FUNCTION_BLOCK FB_LimSwStatusMCS2 IMPLEMENTS I_LimSwStatusMCS2
VAR_INPUT
END_VAR
VAR_OUTPUT
END_VAR
VAR
    bPositiveDirection : BOOL;
    bNegativeDirection : BOOL;
    bMoveBackwardEnabled : BOOL;
    bMoveForwardEnabled : BOOL;
    bInternalLimitActive : BOOL;
    bWarningCondition : BOOL;
    bLimOverride : BOOL;
END_VAR

// Read Limits status and update shared space
bMoveBackwardEnabled := bLimOverride OR NOT(THIS^.bNegativeDirection AND ( THIS^.bInternalLimitActive OR THIS^.bWarningCondition ));
bMoveForwardEnabled := bLimOverride OR NOT(THIS^.bPositiveDirection AND ( THIS^.bInternalLimitActive OR THIS^.bWarningCondition ));

METHOD AxisStatus
VAR_INPUT
    PositiveDirection	: BOOL;
    NegativeDirection	: BOOL;
END_VAR
bPositiveDirection:=PositiveDirection;
bNegativeDirection:=NegativeDirection;
END_METHOD

{warning 'Add property implementation'}
PROPERTY InternalLimitActive : BOOL
GET
END_GET
SET
END_SET
END_PROPERTY

METHOD InternalLimits
VAR_INPUT
    InternalLimitActive	: BOOL;
    WarningCondition	: BOOL;
END_VAR
bInternalLimitActive := InternalLimitActive;
bWarningCondition := WarningCondition;
END_METHOD

{warning 'Add property implementation'}
PROPERTY LimBackward : BOOL
GET
END_GET
END_PROPERTY

{warning 'Add property implementation'}
PROPERTY LimForward : BOOL
GET
END_GET
END_PROPERTY

{warning 'Add property implementation'}
PROPERTY LimHome : BOOL
GET
END_GET
END_PROPERTY

{warning 'Add property implementation'}
PROPERTY LimOverride : BOOL
GET
END_GET
SET
END_SET
END_PROPERTY

{warning 'Add property implementation'}
PROPERTY MoveBackwardEnabled : BOOL
GET
END_GET
END_PROPERTY

{warning 'Add property implementation'}
PROPERTY MoveForwardEnabled : BOOL
GET
END_GET
END_PROPERTY

{warning 'Add property implementation'}
PROPERTY WarningCondition : BOOL
GET
END_GET
SET
END_SET
END_PROPERTY

END_FUNCTION_BLOCK

(* stored: Version 1.1.0.1
   POU FB_LimSwStatusMCS2: Id {e82c472b-4e09-459d-83c5-e6524de07cc9}, SpecialFunc None
   Method AxisStatus: Id {b6a43cf8-24d6-42e3-9ffa-0a6a1fcfe0c2}
   Property InternalLimitActive: Id {9785faa9-6e22-4b72-879f-74f38349c993}
   Get Get: Id {d5fc83b0-3602-4b79-b305-31cda962b007}
   Set Set: Id {3ae2133f-fa8c-4126-95ec-f568abc28cb6}
   Method InternalLimits: Id {3d906f1c-4309-4620-b9c2-d5fcc535cf78}
   Property LimBackward: Id {f4561d22-7e93-44a3-9f7c-57ae1fe2e3b3}
   Get Get: Id {cdcf507d-848d-4f9c-811a-85a48621b9c6}
   Property LimForward: Id {ca690340-85a0-4f97-ae9b-9715ca070efc}
   Get Get: Id {1c921a6f-9947-45c2-b6d7-11d1ee5af807}
   Property LimHome: Id {6205f904-d29b-4a41-a324-cb85ab0bac79}
   Get Get: Id {bc24439f-4f81-4ed3-b2a3-e6911e658400}
   Property LimOverride: Id {ceedabb0-daa0-442b-8e15-dce5027b9271}
   Get Get: Id {3a655c80-5eaf-46a0-819e-54f24c5af205}
   Set Set: Id {9f94dc7d-e710-4f23-bc6d-cad3a3c0a365}
   Property MoveBackwardEnabled: Id {eccf17a9-719a-4c3e-be00-13d2ff40a848}
   Get Get: Id {90fc8736-3356-4c91-ad5a-653e31d1f3c7}
   Property MoveForwardEnabled: Id {34a229a6-baa1-4b86-a121-499909debdce}
   Get Get: Id {66284a56-ab30-4db4-a044-8207c4c32f35}
   Property WarningCondition: Id {5cf554e9-711d-44d7-9224-89ae7d59504b}
   Get Get: Id {e4342f9b-0b2d-458c-8725-a74b200c3d69}
   Set Set: Id {25d14368-41f7-4479-8859-3fe91648a99e} *)
